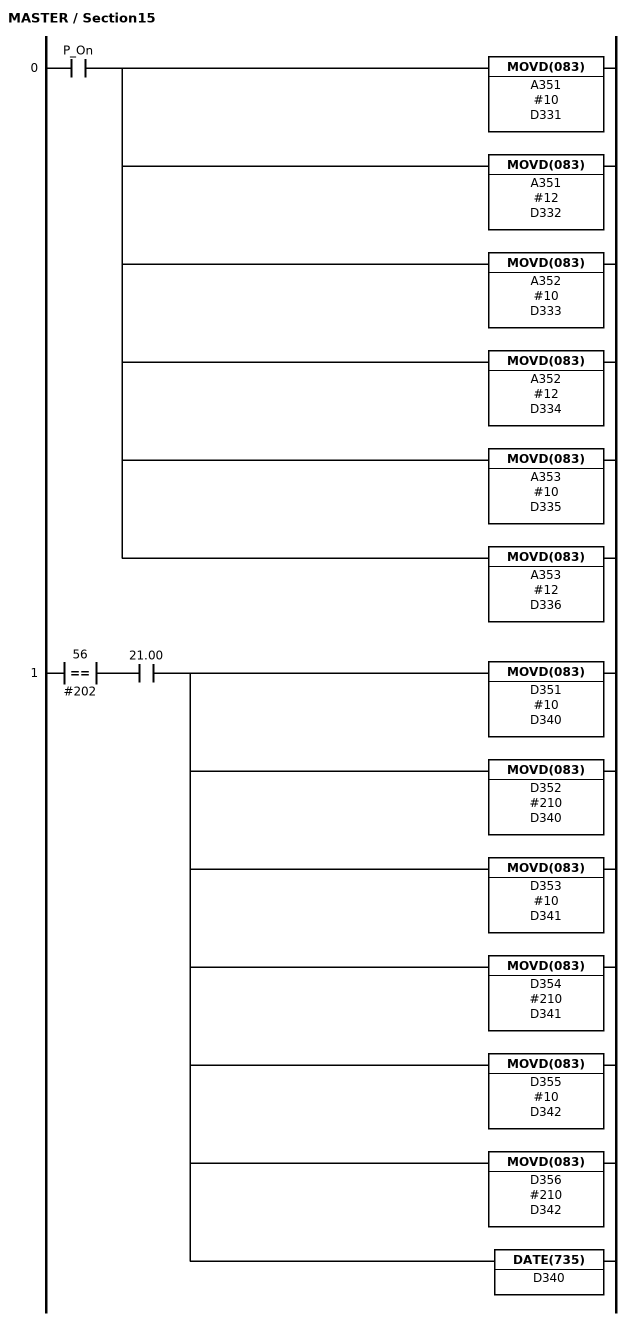
; [picture p72: MASTER / Section15, rungs 0-1]
; rung 0
// R
LD P_On
MOVD(083) A351 #10 D331
MOVD(083) A351 #12 D332
MOVD(083) A352 #10 D333
MOVD(083) A352 #12 D334
MOVD(083) A353 #10 D335
MOVD(083) A353 #12 D336
; rung 1
LD=(300) 56 #202
AND 21.00
MOVD(083) D351 #10 D340
MOVD(083) D352 #210 D340
MOVD(083) D353 #10 D341
MOVD(083) D354 #210 D341
MOVD(083) D355 #10 D342
MOVD(083) D356 #210 D342
DATE(735) D340
; rung 2
END(001)

## Program ZALACZANIE (cyclic task 4)

### Section Section1

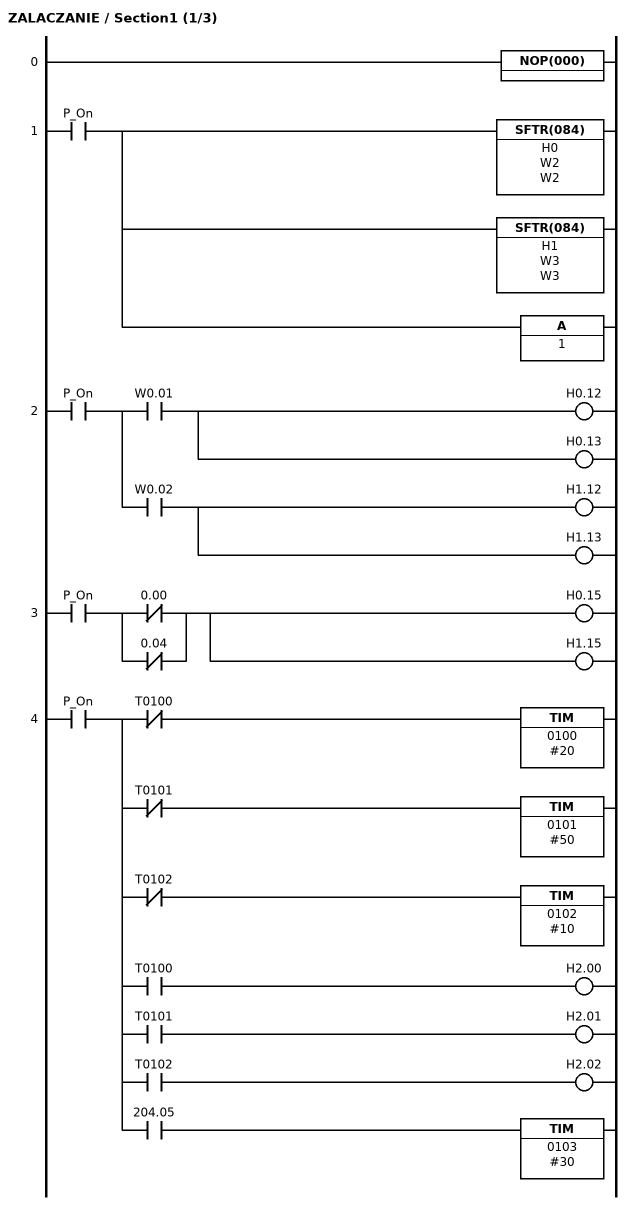
; rung 0
NOP(000)
; rung 1
LD P_On
SFTR(084) H0 W2 W2
SFTR(084) H1 W3 W3  // 
A  1
// 
; rung 2
LD P_On
OUT TR0
AND W0.01
OUT H0.12
OUT H0.13
LD TR0
AND W0.02
OUT H1.12
OUT H1.13
; rung 3
LD P_On
LDNOT 0.00
ORNOT 0.04
ANDLD
OUT H0.15
OUT H1.15
; rung 4
LD P_On
OUT TR0
ANDNOT T0100
TIM 0100 #20
LD TR0
ANDNOT T0101
TIM 0101 #50
LD TR0
ANDNOT T0102
TIM 0102 #10
LD TR0
AND T0100
OUT H2.00
LD TR0
AND T0101
OUT H2.01
LD TR0
AND T0102
OUT H2.02
LD TR0
AND 204.05
TIM 0103 #30

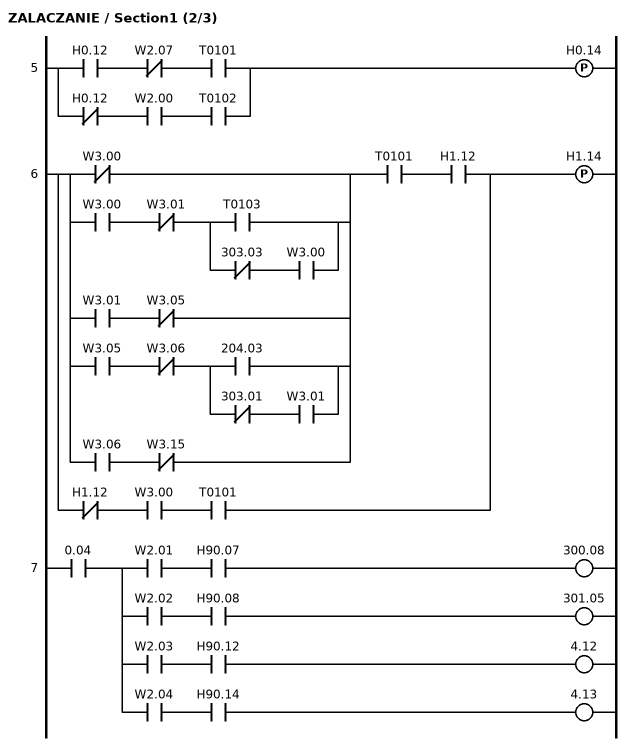
; rung 5
LD H0.12
ANDNOT W2.07
AND T0101
LDNOT H0.12
AND W2.00
AND T0102
ORLD
DIFU(013) H0.14
; rung 6
LDNOT W3.00
LD W3.00
ANDNOT W3.01
LD T0103
LDNOT 303.03
AND W3.00
ORLD
ANDLD
ORLD
LD W3.01
ANDNOT W3.05
ORLD
LD W3.05
ANDNOT W3.06
LD 204.03
LDNOT 303.01
AND W3.01
ORLD
ANDLD
ORLD
LD W3.06
ANDNOT W3.15
ORLD
AND T0101
AND H1.12
LDNOT H1.12
AND W3.00
AND T0101
ORLD
DIFU(013) H1.14
; rung 7
// R
LD 0.04
OUT TR0
AND W2.01
AND H90.07
OUT 300.08
LD TR0
AND W2.02
AND H90.08
OUT 301.05
LD TR0
AND W2.03
AND H90.12
OUT 4.12
LD TR0
AND W2.04
AND H90.14
OUT 4.13

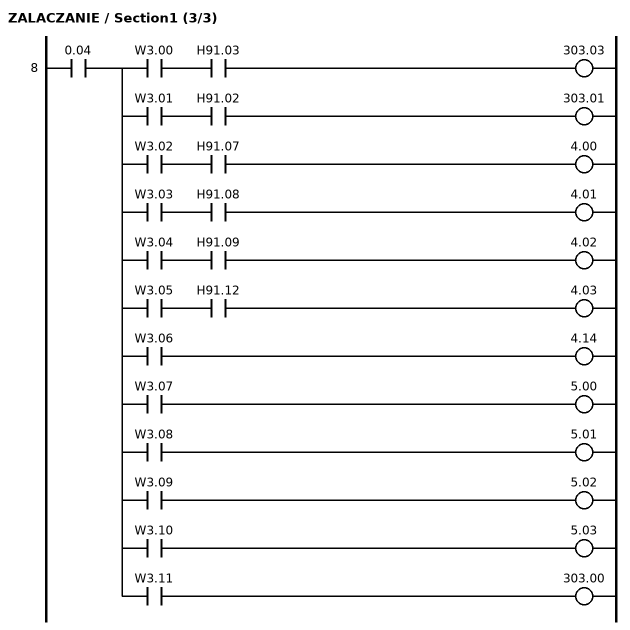
; rung 8
// R
LD 0.04
OUT TR0
AND W3.00
AND H91.03
OUT 303.03
LD TR0
AND W3.01
AND H91.02
OUT 303.01
LD TR0
AND W3.02
AND H91.07
OUT 4.00
LD TR0
AND W3.03
AND H91.08
OUT 4.01
LD TR0
AND W3.04
AND H91.09
OUT 4.02
LD TR0
AND W3.05
AND H91.12
OUT 4.03
LD TR0
AND W3.06
OUT 4.14
LD TR0
AND W3.07
OUT 5.00
LD TR0
AND W3.08
OUT 5.01
LD TR0
AND W3.09
OUT 5.02
LD TR0
AND W3.10
OUT 5.03
LD TR0
AND W3.11
OUT 303.00
; rung 9
END(001)

## Program ASP_FOLIA (cyclic task 5)

### Section Section1

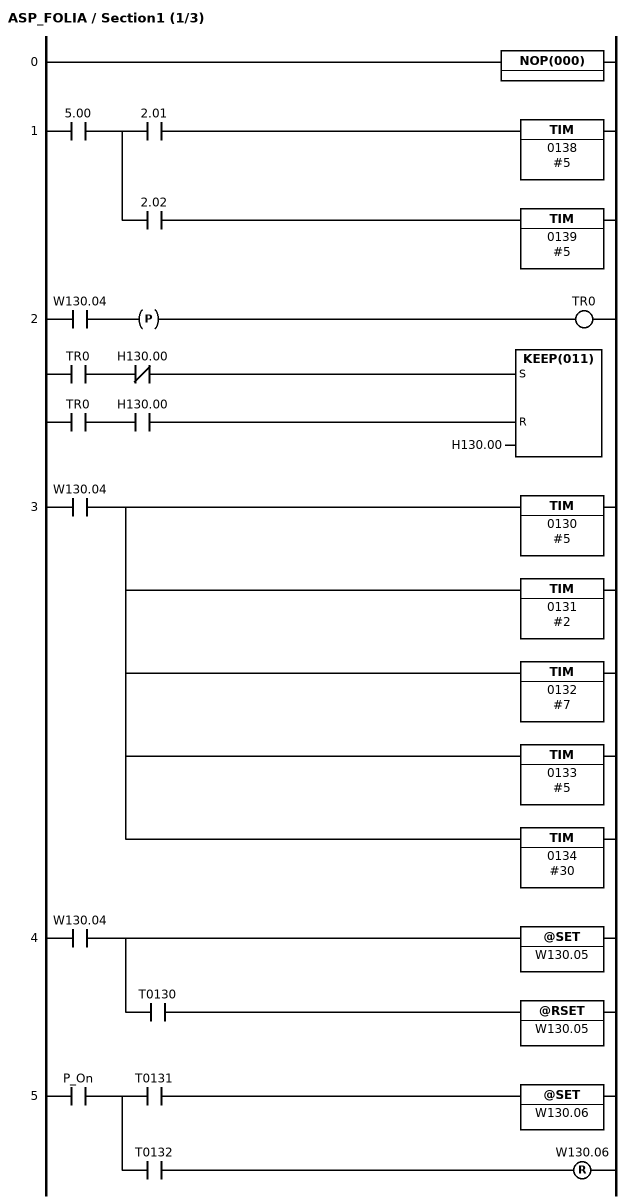
; rung 0
NOP(000)
; rung 1
LD 5.00
OUT TR0
AND 2.01
TIM 0138 #5
LD TR0
AND 2.02
TIM 0139 #5
; rung 2
LD W130.04
UP(521)
OUT TR0
ANDNOT H130.00
LD TR0
AND H130.00
KEEP(011) H130.00
; rung 3
LD W130.04
TIM 0130 #5
TIM 0131 #2
TIM 0132 #7
TIM 0133 #5
TIM 0134 #30
; rung 4
LD W130.04
@SET W130.05
AND T0130
@RSET W130.05
; rung 5
LD P_On
OUT TR0
AND T0131
@SET W130.06
LD TR0
AND T0132
RSET W130.06

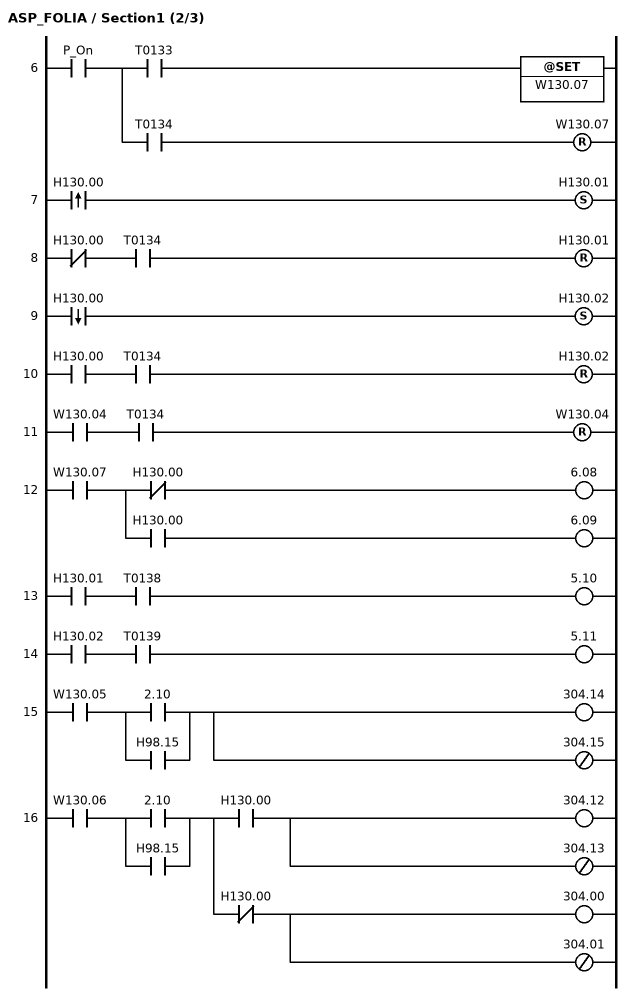
; rung 6
LD P_On
OUT TR0
AND T0133
@SET W130.07
LD TR0
AND T0134
RSET W130.07
; rung 7
@LD H130.00
SET H130.01
; rung 8
LDNOT H130.00
AND T0134
RSET H130.01
; rung 9
%LD H130.00
SET H130.02
; rung 10
LD H130.00
AND T0134
RSET H130.02
; rung 11
LD W130.04
AND T0134
RSET W130.04
; rung 12
LD W130.07
OUT TR0
ANDNOT H130.00
OUT 6.08
LD TR0
AND H130.00
OUT 6.09
; rung 13
LD H130.01
AND T0138
OUT 5.10
; rung 14
LD H130.02
AND T0139
OUT 5.11
; rung 15
LD W130.05
LD 2.10
OR H98.15
ANDLD
OUT 304.14
OUTNOT 304.15
; rung 16
LD W130.06
LD 2.10
OR H98.15
ANDLD
OUT TR0
AND H130.00
OUT 304.12
OUTNOT 304.13
LD TR0
ANDNOT H130.00
OUT 304.00
OUTNOT 304.01

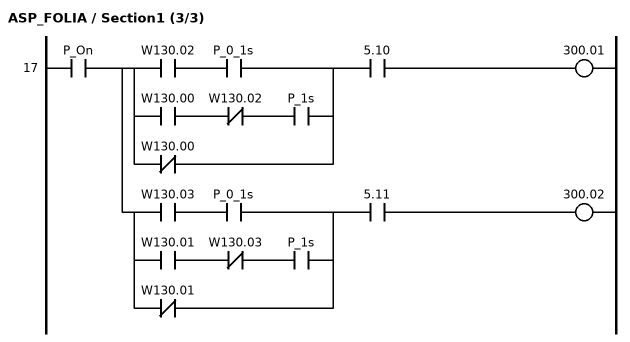
; rung 17
LD P_On
OUT TR0
LD W130.02
AND P_0_1s
LD W130.00
ANDNOT W130.02
AND P_1s
ORLD
ORNOT W130.00
AND 5.10
ANDLD
OUT 300.01
LD TR0
LD W130.03
AND P_0_1s
LD W130.01
ANDNOT W130.03
AND P_1s
ORLD
ORNOT W130.01
AND 5.11
ANDLD
OUT 300.02
; rung 18
END(001)

## Program ASP_WŁÓKNINA (cyclic task 6)

### Section Section1

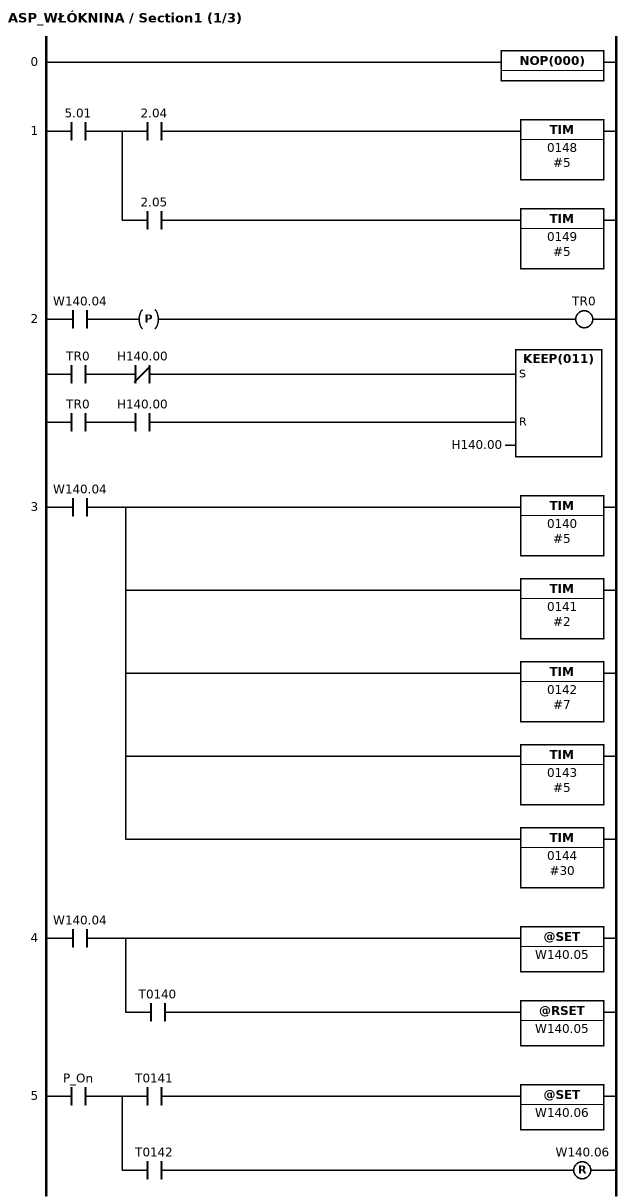
; rung 0
NOP(000)
; rung 1
LD 5.01
OUT TR0
AND 2.04
TIM 0148 #5
LD TR0
AND 2.05
TIM 0149 #5
; rung 2
LD W140.04
UP(521)
OUT TR0
ANDNOT H140.00
LD TR0
AND H140.00
KEEP(011) H140.00
; rung 3
LD W140.04
TIM 0140 #5
TIM 0141 #2
TIM 0142 #7
TIM 0143 #5
TIM 0144 #30
; rung 4
LD W140.04
@SET W140.05
AND T0140
@RSET W140.05
; rung 5
LD P_On
OUT TR0
AND T0141
@SET W140.06
LD TR0
AND T0142
RSET W140.06

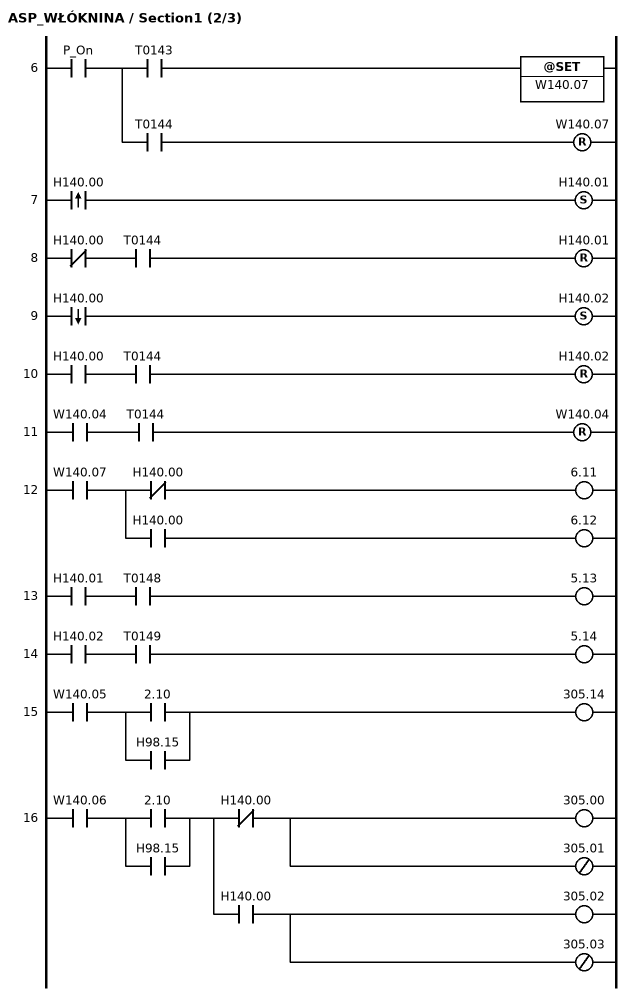
; rung 6
LD P_On
OUT TR0
AND T0143
@SET W140.07
LD TR0
AND T0144
RSET W140.07
; rung 7
@LD H140.00
SET H140.01
; rung 8
LDNOT H140.00
AND T0144
RSET H140.01
; rung 9
%LD H140.00
SET H140.02
; rung 10
LD H140.00
AND T0144
RSET H140.02
; rung 11
LD W140.04
AND T0144
RSET W140.04
; rung 12
LD W140.07
OUT TR0
ANDNOT H140.00
OUT 6.11
LD TR0
AND H140.00
OUT 6.12
; rung 13
LD H140.01
AND T0148
OUT 5.13
; rung 14
LD H140.02
AND T0149
OUT 5.14
; rung 15
LD W140.05
LD 2.10
OR H98.15
ANDLD
OUT 305.14
; rung 16
LD W140.06
LD 2.10
OR H98.15
ANDLD
OUT TR0
ANDNOT H140.00
OUT 305.00
OUTNOT 305.01
LD TR0
AND H140.00
OUT 305.02
OUTNOT 305.03

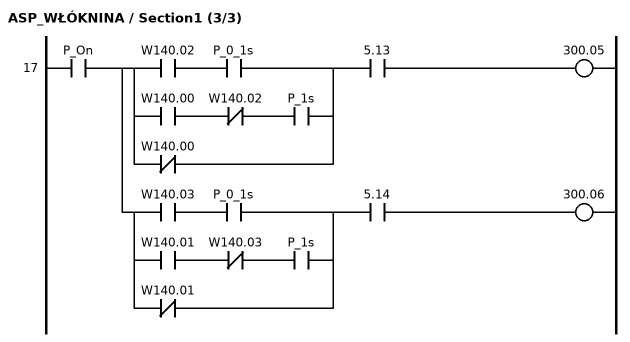
; rung 17
LD P_On
OUT TR0
LD W140.02
AND P_0_1s
LD W140.00
ANDNOT W140.02
AND P_1s
ORLD
ORNOT W140.00
AND 5.13
ANDLD
OUT 300.05
LD TR0
LD W140.03
AND P_0_1s
LD W140.01
ANDNOT W140.03
AND P_1s
ORLD
ORNOT W140.01
AND 5.14
ANDLD
OUT 300.06
; rung 18
END(001)

## Program ASP_PASEK_DL (cyclic task 8)

### Section Section1

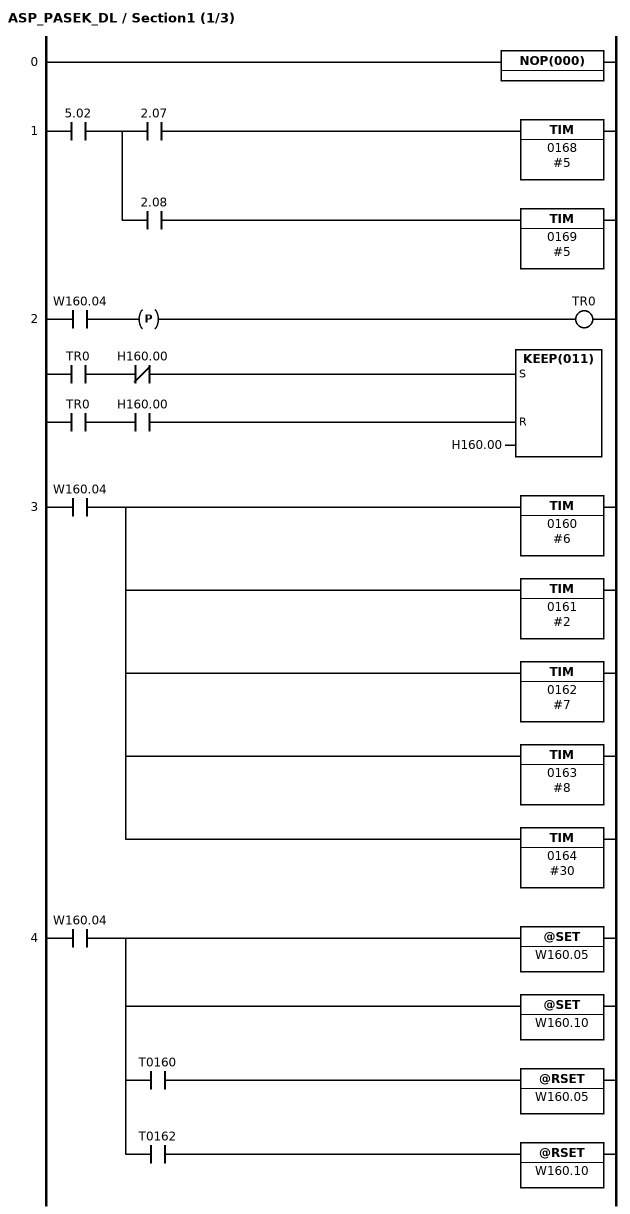
; rung 0
NOP(000)
; rung 1
LD 5.02
OUT TR0
AND 2.07
TIM 0168 #5
LD TR0
AND 2.08
TIM 0169 #5
; rung 2
LD W160.04
UP(521)
OUT TR0
ANDNOT H160.00
LD TR0
AND H160.00
KEEP(011) H160.00
; rung 3
LD W160.04
TIM 0160 #6
TIM 0161 #2
TIM 0162 #7
TIM 0163 #8
TIM 0164 #30
; rung 4
LD W160.04
OUT TR0
@SET W160.05
@SET W160.10
AND T0160
@RSET W160.05
LD TR0
AND T0162
@RSET W160.10

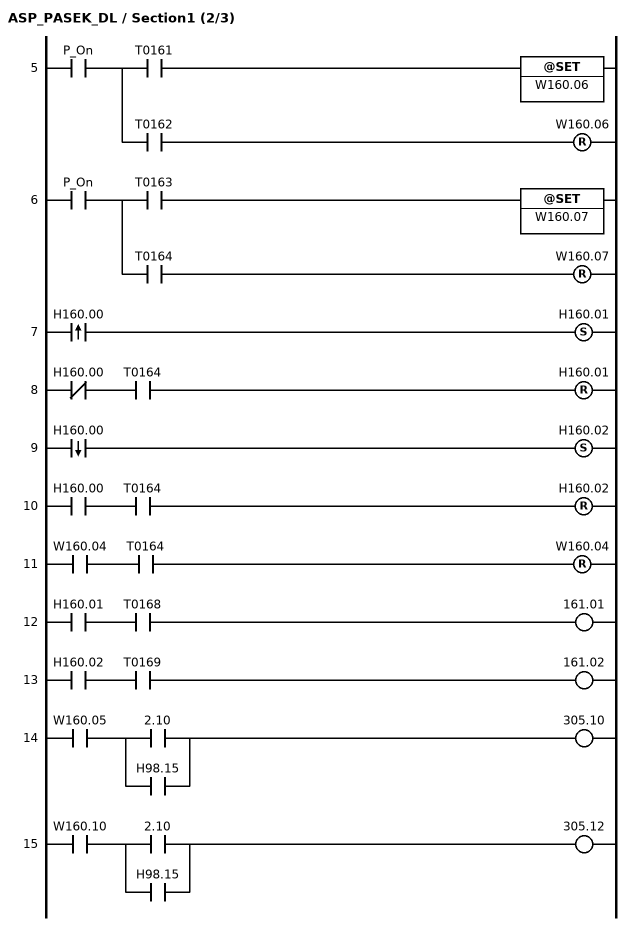
; rung 5
LD P_On
OUT TR0
AND T0161
@SET W160.06
LD TR0
AND T0162
RSET W160.06
; rung 6
LD P_On
OUT TR0
AND T0163
@SET W160.07
LD TR0
AND T0164
RSET W160.07
; rung 7
@LD H160.00
SET H160.01
; rung 8
LDNOT H160.00
AND T0164
RSET H160.01
; rung 9
%LD H160.00
SET H160.02
; rung 10
LD H160.00
AND T0164
RSET H160.02
; rung 11
LD W160.04
AND T0164
RSET W160.04
; rung 12
LD H160.01
AND T0168
OUT 161.01
; rung 13
LD H160.02
AND T0169
OUT 161.02
; rung 14
LD W160.05
LD 2.10
OR H98.15
ANDLD
OUT 305.10
; rung 15
LD W160.10
LD 2.10
OR H98.15
ANDLD
OUT 305.12

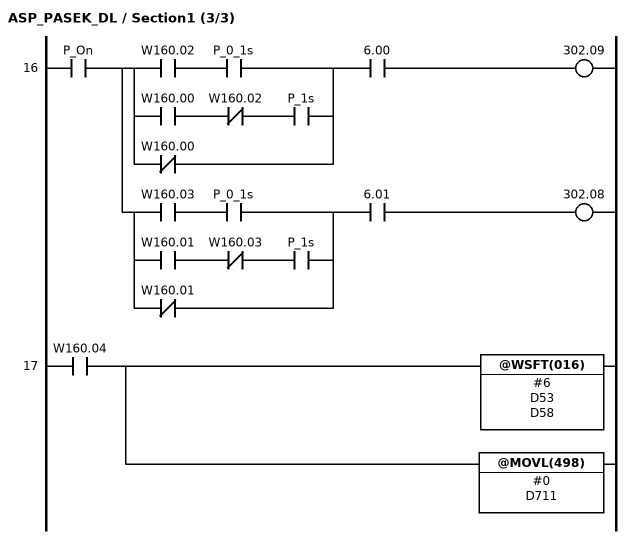
; rung 16
LD P_On
OUT TR0
LD W160.02
AND P_0_1s
LD W160.00
ANDNOT W160.02
AND P_1s
ORLD
ORNOT W160.00
AND 6.00
ANDLD
OUT 302.09
LD TR0
LD W160.03
AND P_0_1s
LD W160.01
ANDNOT W160.03
AND P_1s
ORLD
ORNOT W160.01
AND 6.01
ANDLD
OUT 302.08
; rung 17
LD W160.04
@WSFT(016) #6 D53 D58
@MOVL(498) #0 D711
; rung 18
END(001)

## Program POD_CELULOZY (cyclic task 12)

### Section Section1

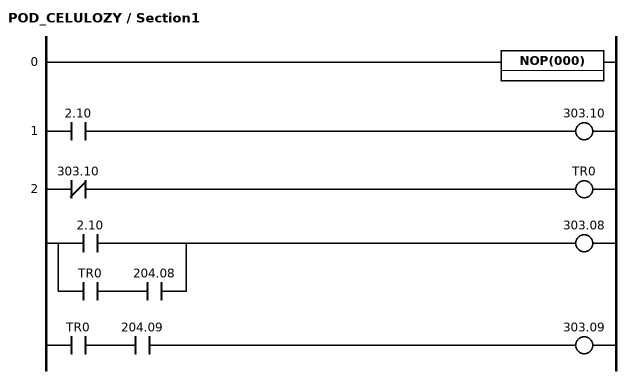
; rung 0
NOP(000)
; rung 1
LD 2.10
OUT 303.10
; rung 2
LD 2.10
LDNOT 303.10
OUT TR0
AND 204.08
ORLD
OUT 303.08
LD TR0
AND 204.09
OUT 303.09

### Section Section2

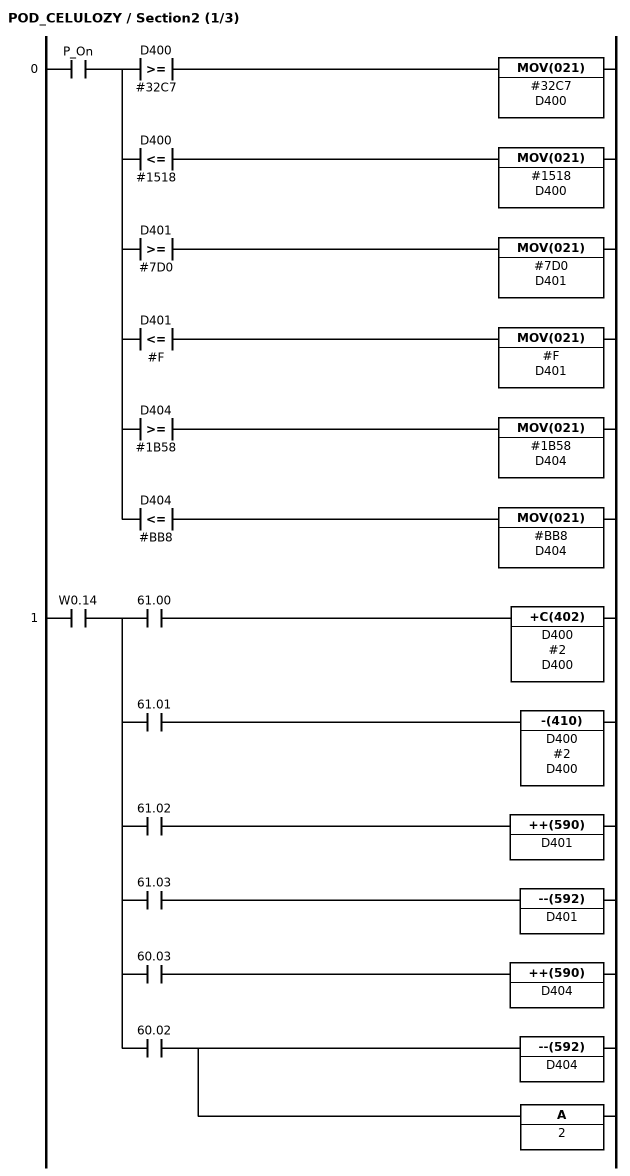
; rung 0
LD P_On
OUT TR0
AND>=(325) D400 #32C7
MOV(021) #32C7 D400
LD TR0
AND<=(315) D400 #1518
MOV(021) #1518 D400
LD TR0
AND>=(325) D401 #7D0
MOV(021) #7D0 D401
LD TR0
AND<=(315) D401 #F
MOV(021) #F D401
LD TR0
AND>=(325) D404 #1B58
MOV(021) #1B58 D404
LD TR0
AND<=(315) D404 #BB8
MOV(021) #BB8 D404
; rung 1
LD W0.14  // 
OUT TR0
AND 61.00
+C(402) D400 #2 D400
LD TR0
AND 61.01
-(410) D400 #2 D400
LD TR0
AND 61.02
++(590) D401
LD TR0
AND 61.03
--(592) D401
LD TR0
AND 60.03
++(590) D404
LD TR0
AND 60.02
--(592) D404  // 
A  2
// 

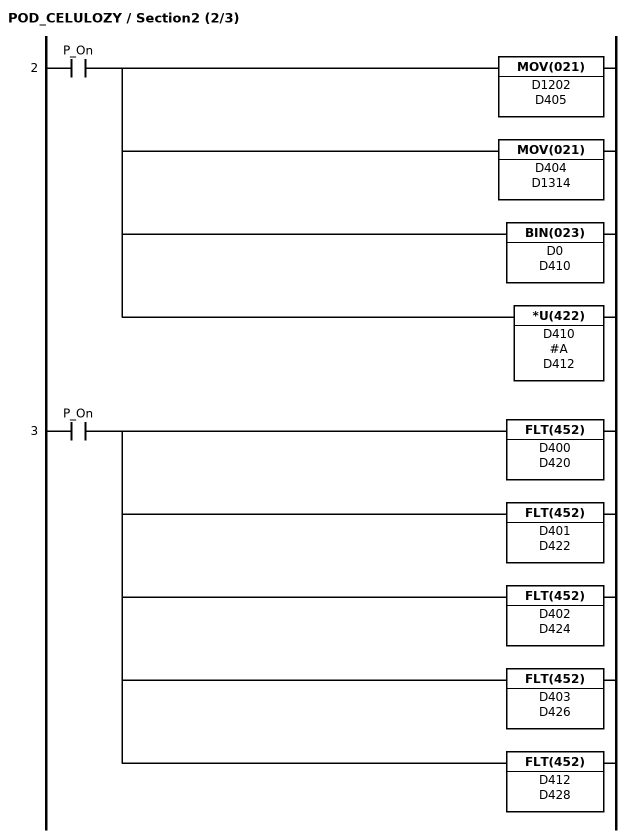
; rung 2
LD P_On
MOV(021) D1202 D405
MOV(021) D404 D1314
BIN(023) D0 D410
*U(422) D410 #A D412
; rung 3
// R
LD P_On
FLT(452) D400 D420
FLT(452) D401 D422
FLT(452) D402 D424
FLT(452) D403 D426
FLT(452) D412 D428

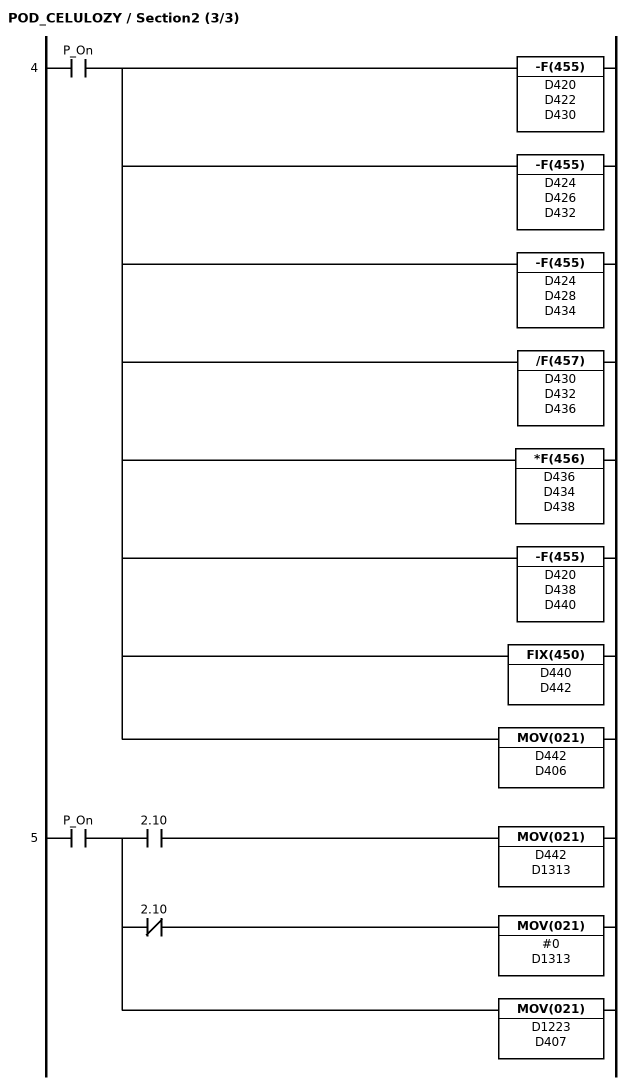
; rung 4
LD P_On
-F(455) D420 D422 D430  // 
-F(455) D424 D426 D432  // 
-F(455) D424 D428 D434  // 
/F(457) D430 D432 D436  // 
*F(456) D436 D434 D438  // 
-F(455) D420 D438 D440
FIX(450) D440 D442
MOV(021) D442 D406
; rung 5
LD P_On
OUT TR0
AND 2.10
MOV(021) D442 D1313
LD TR0
ANDNOT 2.10
MOV(021) #0 D1313
LD TR0
MOV(021) D1223 D407
; rung 6
END(001)

## Program KLEJE (cyclic task 18)

### Section Section1

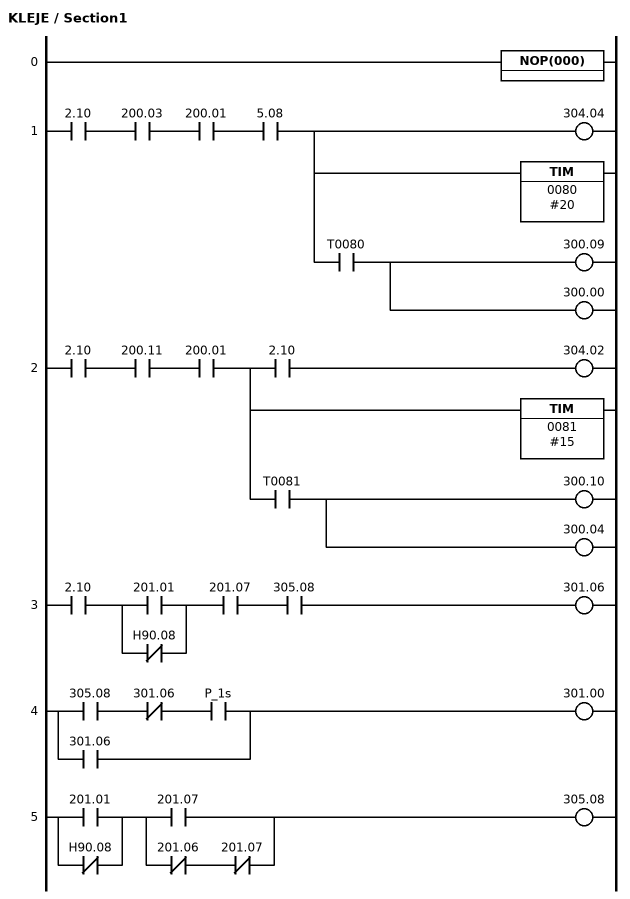
; rung 0
NOP(000)
; rung 1
// R
LD 2.10
AND 200.03
AND 200.01
AND 5.08
OUT 304.04
TIM 0080 #20
AND T0080
OUT 300.09
OUT 300.00
; rung 2
// R
LD 2.10
AND 200.11
AND 200.01
OUT TR0
AND 2.10
OUT 304.02
LD TR0
TIM 0081 #15
AND T0081
OUT 300.10
OUT 300.04
; rung 3
// R
LD 2.10
LD 201.01
ORNOT H90.08
ANDLD
AND 201.07
AND 305.08
OUT 301.06
; rung 4
LD 305.08
ANDNOT 301.06
AND P_1s
OR 301.06
OUT 301.00
; rung 5
LD 201.01
ORNOT H90.08
LD 201.07
LDNOT 201.06
ANDNOT 201.07
ORLD
ANDLD
OUT 305.08
; rung 6
END(001)

## Program OPCJE (cyclic task 19)

### Section Section1

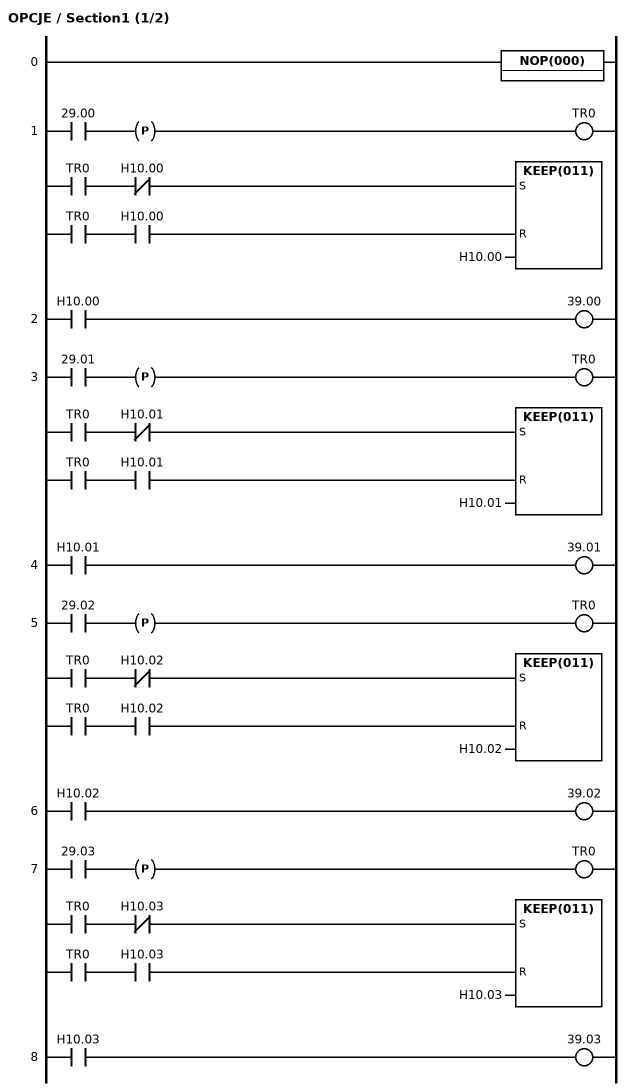
; rung 0
NOP(000)
; rung 1
// R
LD 29.00
UP(521)
OUT TR0
ANDNOT H10.00
LD TR0
AND H10.00
KEEP(011) H10.00
; rung 2
LD H10.00
OUT 39.00
; rung 3
// R
LD 29.01
UP(521)
OUT TR0
ANDNOT H10.01
LD TR0
AND H10.01
KEEP(011) H10.01
; rung 4
LD H10.01
OUT 39.01
; rung 5
// R
LD 29.02
UP(521)
OUT TR0
ANDNOT H10.02
LD TR0
AND H10.02
KEEP(011) H10.02
; rung 6
LD H10.02
OUT 39.02
; rung 7
// R
LD 29.03
UP(521)
OUT TR0
ANDNOT H10.03
LD TR0
AND H10.03
KEEP(011) H10.03
; rung 8
LD H10.03
OUT 39.03

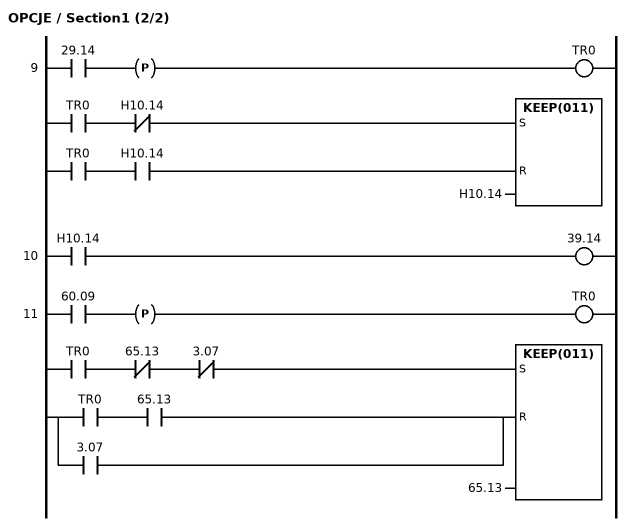
; rung 9
LD 29.14
UP(521)
OUT TR0
ANDNOT H10.14
LD TR0
AND H10.14
KEEP(011) H10.14
; rung 10
LD H10.14
OUT 39.14
; rung 11
LD 60.09
UP(521)
OUT TR0
ANDNOT 65.13
ANDNOT 3.07
LD TR0
AND 65.13
OR 3.07
KEEP(011) 65.13
; rung 12
END(001)

## Program REG_FAZY (cyclic task 20)

### Section Section1

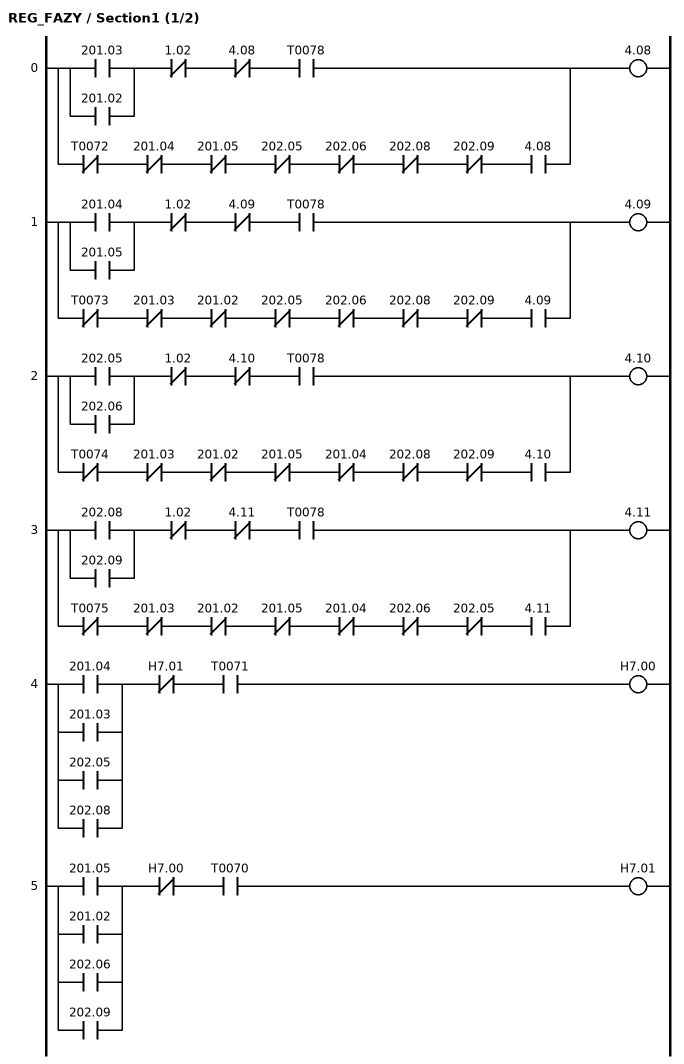
; rung 0
// R
LD 201.03
OR 201.02
ANDNOT 1.02
ANDNOT 4.08
AND T0078
LDNOT T0072
ANDNOT 201.04
ANDNOT 201.05
ANDNOT 202.05
ANDNOT 202.06
ANDNOT 202.08
ANDNOT 202.09
AND 4.08
ORLD
OUT 4.08  // 
; rung 1
LD 201.04
OR 201.05
ANDNOT 1.02
ANDNOT 4.09
AND T0078
LDNOT T0073
ANDNOT 201.03
ANDNOT 201.02
ANDNOT 202.05
ANDNOT 202.06
ANDNOT 202.08
ANDNOT 202.09
AND 4.09
ORLD
OUT 4.09  // 
; rung 2
LD 202.05
OR 202.06
ANDNOT 1.02
ANDNOT 4.10
AND T0078
LDNOT T0074
ANDNOT 201.03
ANDNOT 201.02
ANDNOT 201.05
ANDNOT 201.04
ANDNOT 202.08
ANDNOT 202.09
AND 4.10
ORLD
OUT 4.10  // 
; rung 3
LD 202.08
OR 202.09
ANDNOT 1.02
ANDNOT 4.11
AND T0078
LDNOT T0075
ANDNOT 201.03
ANDNOT 201.02
ANDNOT 201.05
ANDNOT 201.04
ANDNOT 202.06
ANDNOT 202.05
AND 4.11
ORLD
OUT 4.11  // 
; rung 4
LD 201.04
OR 201.03
OR 202.05
OR 202.08
ANDNOT H7.01
AND T0071
OUT H7.00
; rung 5
LD 201.05
OR 201.02
OR 202.06
OR 202.09
ANDNOT H7.00
AND T0070
OUT H7.01

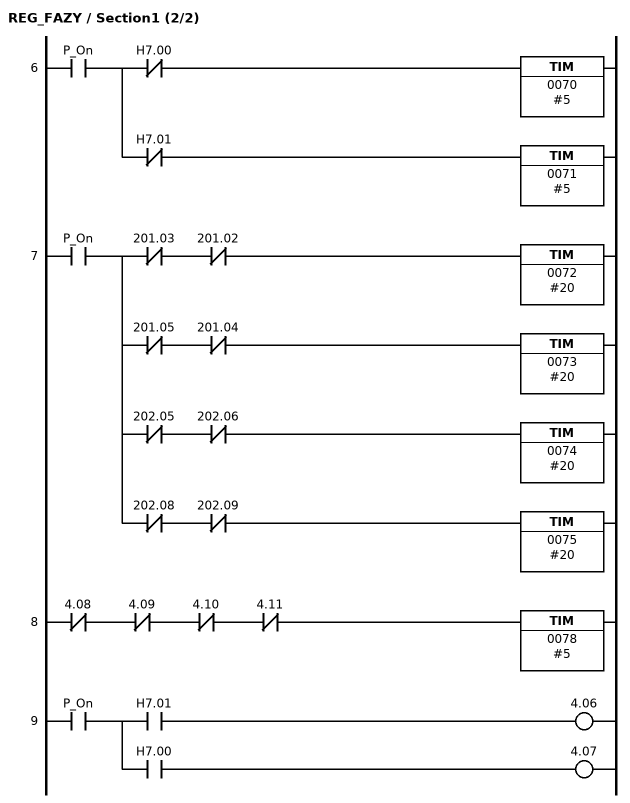
; rung 6
LD P_On
OUT TR0
ANDNOT H7.00
TIM 0070 #5
LD TR0
ANDNOT H7.01
TIM 0071 #5
; rung 7
LD P_On
OUT TR0
ANDNOT 201.03
ANDNOT 201.02
TIM 0072 #20
LD TR0
ANDNOT 201.05
ANDNOT 201.04
TIM 0073 #20
LD TR0
ANDNOT 202.05
ANDNOT 202.06
TIM 0074 #20
LD TR0
ANDNOT 202.08
ANDNOT 202.09
TIM 0075 #20
; rung 8
LDNOT 4.08
ANDNOT 4.09
ANDNOT 4.10
ANDNOT 4.11
TIM 0078 #5
; rung 9
LD P_On
OUT TR0
AND H7.01
OUT 4.06
LD TR0
AND H7.00
OUT 4.07  // 
; rung 10
END(001)

## Program ZMIANA_1 (cyclic task 21)

### Section Section1

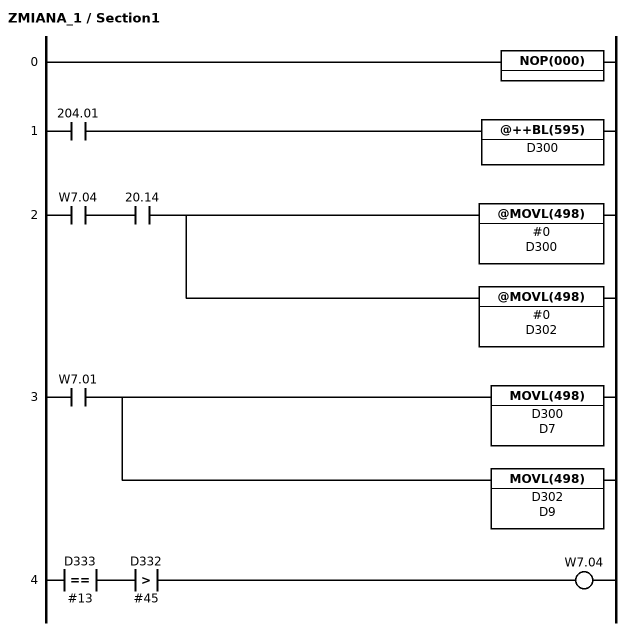
; rung 0
NOP(000)
; rung 1
LD 204.01
@++BL(595) D300
; rung 2
LD W7.04
AND 20.14
@MOVL(498) #0 D300
@MOVL(498) #0 D302
; rung 3
LD W7.01
MOVL(498) D300 D7
MOVL(498) D302 D9
; rung 4
LD=(300) D333 #13
AND>(320) D332 #45
OUT W7.04
; rung 5
END(001)

## Program ZMIANA_2 (cyclic task 22)

### Section Section1

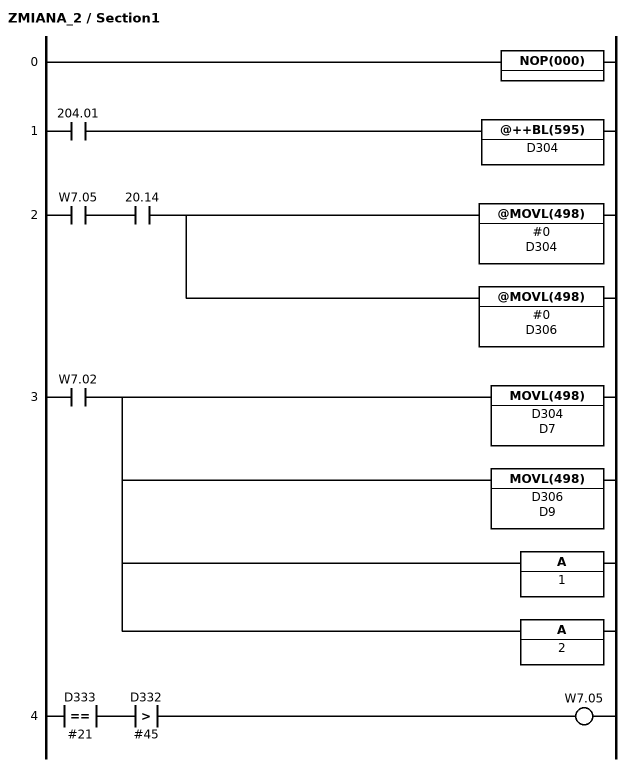
; rung 0
NOP(000)
; rung 1
LD 204.01
@++BL(595) D304
; rung 2
LD W7.05
AND 20.14
@MOVL(498) #0 D304
@MOVL(498) #0 D306
; rung 3
LD W7.02
MOVL(498) D304 D7
MOVL(498) D306 D9  // 
A  1
A  2
// 
// 
; rung 4
LD=(300) D333 #21
AND>(320) D332 #45
OUT W7.05
; rung 5
END(001)

## Program ZMIANA_3 (cyclic task 23)

### Section Section1

